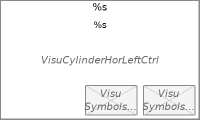
VISUALIZATION VisuCylinderHorLeft  // 200x120
VAR_IN_OUT
	fbVisuCylinder: FB_VISU_CYLINDER;
END_VAR
    Textfield (0,15 200x20), "%s", text variable: fbVisuCylinder.strInfo, colour toggle: fbVisuCylinder.stEvent.bEventActive
    Textfield (0,0 200x14), "%s", text variable: fbVisuCylinder.strFullObjName
    Image (143,85 52x30), invisible if: fbVisuCylinder.bBaseArrowInvisible, image: VisuSymbols.Symbols.ArrowBoldRight
        p2175578022: fbVisuCylinder.dwFrameColorBase
    Image (85,85 52x30), invisible if: fbVisuCylinder.bWorkArrowInvisible, image: VisuSymbols.Symbols.ArrowBoldLeft
        p2175578022: fbVisuCylinder.dwFrameColorWork
    Group (90,35 105x40)
        p3560616238: fbVisuCylinder.iMove
        RoundedRectangle (-10,10 100x20)
        RoundedRectangle (80,0 20x40)
    Rectangle (85,35 105x40)
        OnMouseClick: execute { fbVisuCylinder.bFrameInvisible:=false; }
    Frame (0,0 200x120), invisible if: fbVisuCylinder.bFrameInvisible, frame switch variable: fbVisuCylinder.iFrame
        shows VisuCylinderHorLeftCtrl(fbVisuCylinder := fbVisuCylinder)
END_VISUALIZATION

(* stored: Version 1.1.0.1, ProductVersion 3.1.4024.12
   Visu VisuCylinderHorLeft: Id {de89adac-0653-462a-9168-c5f7e8a20ba5} *)
